Fanuc KAREL source: kd00055.KL

-- PROVISIONAL review KL for V770-1; original PC SHA256 2d28b74abc44dc49e3ddbaf177aba7a8da4425d10528ffa05c13208c7211e2cd
-- Incomplete behavior may be omitted. Consult companion uncertainty JSON. Do not deploy.
PROGRAM KD00055
%NOLOCKGROUP
VAR
  I : INTEGER
  J : INTEGER
  B : BOOLEAN
  R : REAL
  S : STRING[80]
BEGIN
  -- UNRESOLVED_PC offsets 5-25; opcodes 9D,81,18,9D,1B,9D,12,2E,1B,9D,13,04
  -- UNRESOLVED_PC offsets 30-34; opcodes 7F
END KD00055
